// TIA Portal project "Ampelanlage" (V16)

(* hardware
DEVICE "S71500/ET200MP-Station_1"  S7-1500 station
   slot 0: "Profilschiene_0"  Rack  6ES7 590-1***0-0AA0
   slot 1: "PLC_1"  CPU 1516-3 PN/DP  6ES7 516-3AN02-0AB0  V2.8
      slot 3: "CPU-Display_1"  6ES7591-1BA00-0AA0
      slot 32768: "PROFINET-Schnittstelle_1"  X1
         slot 32769: "Port_1"  X1 P1
         slot 32770: "Port_2"  X1 P2
      slot 33024: "PROFINET-Schnittstelle_2"  X2
         slot 33025: "Port_1"  X2 P1
      slot 33280: "DP-Schnittstelle_1"  X3
      slot 34817: "Virtual CP interface port_1"  Virtual CP interface port  Virtual CP interface port
   slot 2: "DI 32x24VDC HF_1"  DI 32x24VDC HF  6ES7 521-1BL00-0AB0  V2.2
   slot 3: "DQ 32x24VDC/0.5A HF_1"  DQ 32x24VDC/0.5A HF  6ES7 522-1BL01-0AB0  V1.1
   slot 4: "AI 8xU/I/RTD/TC ST_1"  AI 8xU/I/RTD/TC ST  6ES7 531-7KF00-0AB0  V2.2
   slot 5: "AQ 4xU/I ST_1"  AQ 4xU/I ST  6ES7 532-5HD00-0AB0  V2.2
DEVICE "ET 200SP-Station_1"  ET 200SP-Station
   slot 0: "Baugruppenträger_0"  Rack  6ES5 710-8MAx1
   slot 0: "IO-Device_1"  IM 155-6 PN/2 HF  6ES7 155-6AU01-0CN0  V4.2
   slot 1: "DI 8x24VDC HF_1"  DI 8x24VDC HF  6ES7 131-6BF00-0CA0  V2.0
      slot 1: "DI 8x24VDC HF_1"  DI 8x24VDC HF
   slot 2: "DQ 8x24VDC/0.5A HF_1"  DQ 8x24VDC/0.5A HF  6ES7 132-6BF00-0CA0  V2.0
      slot 1: "DQ 8x24VDC/0.5A HF_1"  DQ 8x24VDC/0.5A HF
   slot 3: "AI 2xU/I 2-,4-wire HF_1"  AI 2xU/I 2-,4-wire HF  6ES7 134-6HB00-0CA1  V2.0
      slot 1: "AI 2xU/I 2-,4-wire HF_1"  AI 2xU/I 2-,4-wire HF
   slot 4: "AQ 2xU/I HF_1"  AQ 2xU/I HF  6ES7 135-6HB00-0CA1  V1.0
      slot 1: "AQ 2xU/I HF_1"  AQ 2xU/I HF
   slot 5: "Servermodul_1"  Server module  6ES7 193-6PA00-0AA0  V1.1
      slot 1: "Servermodul_1"  Server module
   slot 127: "BA 2xRJ45"  BA 2xRJ45  6ES7 193-6AR00-0AA0  V0.0
      slot 1: "Port_1"  X1 P1 R  6ES7 193-6AR00-0AA0  V0.0
      slot 2: "Port_2"  X1 P2 R  6ES7 193-6AR00-0AA0  V0.0
*)

// ===== PLC "PLC_1"  CPU 1516-3 PN/DP =====

VAR_GLOBAL   // PLC tag table "Ampelanlage"
   "xS0" AT %I0.0 : Bool;   // Anlage aus
   "xS7" AT %I0.7 : Bool;   // Anlage ein
   "xH0" AT %Q0.0 : Bool;   // Rot Hauptstraße
   "xH1" AT %Q0.1 : Bool;   // Gelb Hauptstraße
   "xH2" AT %Q0.2 : Bool;   // Grün Hauptsraße
   "xH3" AT %Q0.3 : Bool;   // Rot Nebenstraße
   "xH4" AT %Q0.4 : Bool;   // Gelb Nebenstraße
   "xH5" AT %Q0.5 : Bool;   // Grün Nebenstraße
   "xH6" AT %Q0.6 : Bool;   // Rot Fußgängerüberrweg
   "xH7" AT %Q0.7 : Bool;   // Grün Fußgängerüberweg
   "xS1" AT %I0.1 : Bool;   // S1 Haupt
   "xS2" AT %I0.2 : Bool;   // S2 Haupt
   "xS3" AT %I0.3 : Bool;   // S3 Neben
   "xS5" AT %I0.5 : Bool;   // S5 Fuß
   "xS6" AT %I0.6 : Bool;   // S6 Fuß
END_VAR

DATA_BLOCK "fb_Ampelanlage_DB"   // DB1
{ S7_Optimized_Access := 'TRUE' }
VERSION : 0.1
// stored: InstanceOfName fb_Ampelanlage
"fb_Ampelanlage"
BEGIN
END_DATA_BLOCK

DATA_BLOCK "fb_Ampelanlage_Bodenkontakt_DB"   // DB2
{ S7_Optimized_Access := 'TRUE' }
VERSION : 0.1
// stored: InstanceOfName fb_Ampelanlage_Bodenkontakt
"fb_Ampelanlage_Bodenkontakt"
BEGIN
END_DATA_BLOCK

FUNCTION_BLOCK "fb_Ampelanlage"   // FB1, GRAPH_PLUS
{ S7_Optimized_Access := 'TRUE' }
VERSION : 0.1
   VAR_INPUT
      OFF_SQ : Bool := false;   // Kette ausschalten
      INIT_SQ : Bool := false;   // Kette in Initialzustand versetzen
      ACK_EF : Bool := false;   // Alle Fehler und Störungen quittieren
      S_PREV : Bool := false;   // Vorherigen Schritt am Parameter S_NO ausgeben
      S_NEXT : Bool := false;   // Nächsten Schritt am Parameter S_NO anzeigen
      SW_AUTO : Bool := false;   // Automatischer Betrieb
      SW_TAP : Bool := false;   // Halbautomatisch/Weiterschalten mit Transition
      SW_TOP : Bool := false;   // Halbautomatisch/Ignoriere Transition
      SW_MAN : Bool := false;   // Handbetrieb
      S_SEL : Int := 0;   // Schritt auswählen, der an S_NO ausgegeben werden soll
      S_ON : Bool := false;   // Schritt aktivieren, der an Parameter S_NO anliegt
      S_OFF : Bool := false;   // Schritt deaktivieren, der an Parameter S_NO anliegt
      T_PUSH : Bool := false;   // Schaltfreigabe für Transition im halbautomatischen Betrieb
   END_VAR
   VAR_OUTPUT
      S_NO : Int := 0;   // Schrittnummer
      S_MORE : Bool := false;   // Weitere Schritte sind vorhanden und können in S_NO angezeigt werden.
      S_ACTIVE : Bool := false;   // Schritt, der an Parameter S_NO angezeigt wird, ist aktiv
      ERR_FLT : Bool := false;   // Sammelfehler Interlock oder Supervision
      AUTO_ON : Bool := false;   // Automatischer Betrieb eingeschaltet
      TAP_ON : Bool := false;   // Halbautomatischer Betrieb/Schritt mit Transition eingeschaltet
      TOP_ON : Bool := false;   // Halbautomatischer Betrieb/Ignoriere Transition eingeschaltet
      MAN_ON : Bool := false;   // Handbetrieb eingeschaltet
   END_VAR
   VAR
      "xTimer T1" : Bool;   // Zeit abgelaufen
      "xTimer T2" : Bool;
      "xTimer T3" : Bool;
      "xTimer T4" : Bool;
      "xTimer T5" : Bool;
      "xTimer T6" : Bool;
      "xTimer T7" : Bool;
      "xTimer T8" : Bool;
      "xTimer T9" : Bool;
      "xTimer T10" : Bool;
      HMI_INFO : Array[0..8] of UInt;
      IF_PAR : G7_IfParPlus_V6;
      RT_DATA : G7_RTDataPlus_V6;   // Interner Datenbereich
      Trans1 : G7_TransitionPlus_V6;   // Transitionsstruktur
      Trans2 : G7_TransitionPlus_V6;   // Transitionsstruktur
      Trans3 : G7_TransitionPlus_V6;   // Transitionsstruktur
      Trans4 : G7_TransitionPlus_V6;   // Transitionsstruktur
      Trans5 : G7_TransitionPlus_V6;   // Transitionsstruktur
      Trans6 : G7_TransitionPlus_V6;   // Transitionsstruktur
      Trans7 : G7_TransitionPlus_V6;   // Transitionsstruktur
      Trans8 : G7_TransitionPlus_V6;   // Transitionsstruktur
      Trans9 : G7_TransitionPlus_V6;   // Transitionsstruktur
      Step1 : G7_StepPlus_V6;   // Schrittstruktur
      Step2 : G7_StepPlus_V6;   // Schrittstruktur
      Step3 : G7_StepPlus_V6;   // Schrittstruktur
      Step4 : G7_StepPlus_V6;   // Schrittstruktur
      Step5 : G7_StepPlus_V6;   // Schrittstruktur
      Step6 : G7_StepPlus_V6;   // Schrittstruktur
      Step7 : G7_StepPlus_V6;   // Schrittstruktur
      Step8 : G7_StepPlus_V6;   // Schrittstruktur
      Step9 : G7_StepPlus_V6;   // Schrittstruktur
      SINI : Array[0..1] of USInt;
      LSTT : Array[0..8] of USInt;
      ATAJ : Array[0..8] of USInt;
      ATAB : Array[0..8] of USInt;
      PSTT : Array[0..8] of USInt;
      NSTT : Array[0..8] of USInt;
      ASSJ : Array[0..8] of USInt;
      ASSB : Array[0..8] of USInt;
      PTTS : Array[0..8] of USInt;
      NTTS : Array[0..8] of USInt;
      SW_SQTS : Array[0..8] of USInt;
      SWITCH : Array[0..0] of USInt;
      TVX : Array[0..1] of USInt;
      TTX : Array[0..1] of USInt;
      TSX : Array[0..1] of USInt;
      S00X : Array[0..1] of USInt;
      SOFFX : Array[0..1] of USInt;
      SONX : Array[0..1] of USInt;
      SAX : Array[0..1] of USInt;
      SERRX : Array[0..9] of USInt;
      SMX : Array[0..9] of USInt;
      S0X : Array[0..9] of USInt;
      S1X : Array[0..9] of USInt;
      IL_ALARM_INST : Diag_Alarm;
      SUP_ALARM_INST : Diag_Alarm;
      STEP_TIME_ALARM_INST : Diag_Alarm;
      IEC_TIMER_INST : IEC_TIMER;
      TRANSACTION_FLAG : Bool := false;
   END_VAR
   // SINI[0] := 2;
   // LSTT[0] := 255;
   // LSTT[1] := 255;
   // LSTT[2] := 255;
   // LSTT[3] := 255;
   // LSTT[4] := 255;
   // LSTT[5] := 255;
   // LSTT[6] := 255;
   // LSTT[7] := 255;
   // ATAJ[1] := 1;
   // ATAJ[2] := 2;
   // ATAJ[3] := 3;
   // ATAJ[4] := 4;
   // ATAJ[5] := 5;
   // ATAJ[6] := 6;
   // ATAJ[7] := 7;
   // ATAJ[8] := 8;
   // ATAB[1] := 1;
   // ATAB[2] := 2;
   // ATAB[3] := 3;
   // ATAB[4] := 4;
   // ATAB[5] := 5;
   // ATAB[6] := 6;
   // ATAB[7] := 7;
   // ATAB[8] := 8;
   // PSTT[1] := 1;
   // PSTT[2] := 2;
   // PSTT[3] := 3;
   // PSTT[4] := 4;
   // PSTT[5] := 5;
   // PSTT[6] := 6;
   // PSTT[7] := 7;
   // PSTT[8] := 8;
   // NSTT[0] := 1;
   // NSTT[1] := 2;
   // NSTT[2] := 3;
   // NSTT[3] := 4;
   // NSTT[4] := 5;
   // NSTT[5] := 6;
   // NSTT[6] := 7;
   // NSTT[7] := 8;
   // ASSJ[1] := 1;
   // ASSJ[2] := 2;
   // ASSJ[3] := 3;
   // ASSJ[4] := 4;
   // ASSJ[5] := 5;
   // ASSJ[6] := 6;
   // ASSJ[7] := 7;
   // ASSJ[8] := 8;
   // ASSB[1] := 1;
   // ASSB[2] := 2;
   // ASSB[3] := 3;
   // ASSB[4] := 4;
   // ASSB[5] := 5;
   // ASSB[6] := 6;
   // ASSB[7] := 7;
   // ASSB[8] := 8;
   // PTTS[0] := 255;
   // PTTS[2] := 1;
   // PTTS[3] := 2;
   // PTTS[4] := 3;
   // PTTS[5] := 4;
   // PTTS[6] := 5;
   // PTTS[7] := 6;
   // PTTS[8] := 7;
   // NTTS[1] := 1;
   // NTTS[2] := 2;
   // NTTS[3] := 3;
   // NTTS[4] := 4;
   // NTTS[5] := 5;
   // NTTS[6] := 6;
   // NTTS[7] := 7;
   // NTTS[8] := 8;
   // TVX[0] := 16#1;
   // TTX[0] := 16#1;
   // TSX[0] := 16#1;
   // S00X[0] := 16#1;
   // SOFFX[0] := 16#1;
   // SONX[0] := 16#1;
   // SAX[0] := 16#1;
   // SERRX[0] := 16#1;
   // SMX[0] := 16#1;
   // S0X[0] := 16#1;
   // S1X[0] := 16#1;
BEGIN
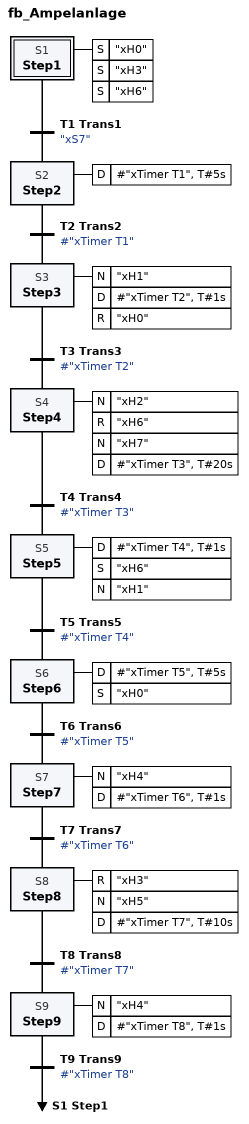
   // sequencer 1
   INITIAL_STEP Step1:   // S1, max time T#10S, warning time T#7S
      // Alle Ampeln Rot
              S    "xH0"
              S    "xH3"
              S    "xH6"
   END_STEP
   TRANSITION Trans1 FROM Step1 TO Step2   // T1
      := "xS7";
   END_TRANSITION
   STEP Step2:   // S2, max time T#10S, warning time T#7S
              D    #"xTimer T1", T#5s
   END_STEP
   TRANSITION Trans2 FROM Step2 TO Step3   // T2
      := #"xTimer T1";
   END_TRANSITION
   STEP Step3:   // S3, max time T#10S, warning time T#7S
              N    "xH1"
              D    #"xTimer T2", T#1s
              R    "xH0"
   END_STEP
   TRANSITION Trans3 FROM Step3 TO Step4   // T3
      := #"xTimer T2";
   END_TRANSITION
   STEP Step4:   // S4, max time T#10S, warning time T#7S
              N    "xH2"
              R    "xH6"
              N    "xH7"
              D    #"xTimer T3", T#20s
   END_STEP
   TRANSITION Trans4 FROM Step4 TO Step5   // T4
      := #"xTimer T3";
   END_TRANSITION
   STEP Step5:   // S5, max time T#10S, warning time T#7S
              D    #"xTimer T4", T#1s
              S    "xH6"
              N    "xH1"
   END_STEP
   TRANSITION Trans5 FROM Step5 TO Step6   // T5
      := #"xTimer T4";
   END_TRANSITION
   STEP Step6:   // S6, max time T#10S, warning time T#7S
              D    #"xTimer T5", T#5s
              S    "xH0"
   END_STEP
   TRANSITION Trans6 FROM Step6 TO Step7   // T6
      := #"xTimer T5";
   END_TRANSITION
   STEP Step7:   // S7, max time T#10S, warning time T#7S
              N    "xH4"
              D    #"xTimer T6", T#1s
   END_STEP
   TRANSITION Trans7 FROM Step7 TO Step8   // T7
      := #"xTimer T6";
   END_TRANSITION
   STEP Step8:   // S8, max time T#10S, warning time T#7S
              R    "xH3"
              N    "xH5"
              D    #"xTimer T7", T#10s
   END_STEP
   TRANSITION Trans8 FROM Step8 TO Step9   // T8
      := #"xTimer T7";
   END_TRANSITION
   STEP Step9:   // S9, max time T#10S, warning time T#7S
              N    "xH4"
              D    #"xTimer T8", T#1s
   END_STEP
   TRANSITION Trans9 FROM Step9 TO Step1   // T9, jump
      := #"xTimer T8";
   END_TRANSITION
END_FUNCTION_BLOCK

FUNCTION_BLOCK "fb_Ampelanlage_Bodenkontakt"   // FB2, GRAPH_PLUS
{ S7_Optimized_Access := 'TRUE' }
VERSION : 0.1
   VAR_INPUT
      OFF_SQ : Bool := false;   // Kette ausschalten
      INIT_SQ : Bool := false;   // Kette in Initialzustand versetzen
      ACK_EF : Bool := false;   // Alle Fehler und Störungen quittieren
      S_PREV : Bool := false;   // Vorherigen Schritt am Parameter S_NO ausgeben
      S_NEXT : Bool := false;   // Nächsten Schritt am Parameter S_NO anzeigen
      SW_AUTO : Bool := false;   // Automatischer Betrieb
      SW_TAP : Bool := false;   // Halbautomatisch/Weiterschalten mit Transition
      SW_TOP : Bool := false;   // Halbautomatisch/Ignoriere Transition
      SW_MAN : Bool := false;   // Handbetrieb
      S_SEL : Int := 0;   // Schritt auswählen, der an S_NO ausgegeben werden soll
      S_ON : Bool := false;   // Schritt aktivieren, der an Parameter S_NO anliegt
      S_OFF : Bool := false;   // Schritt deaktivieren, der an Parameter S_NO anliegt
      T_PUSH : Bool := false;   // Schaltfreigabe für Transition im halbautomatischen Betrieb
   END_VAR
   VAR_OUTPUT
      S_NO : Int := 0;   // Schrittnummer
      S_MORE : Bool := false;   // Weitere Schritte sind vorhanden und können in S_NO angezeigt werden.
      S_ACTIVE : Bool := false;   // Schritt, der an Parameter S_NO angezeigt wird, ist aktiv
      ERR_FLT : Bool := false;   // Sammelfehler Interlock oder Supervision
      AUTO_ON : Bool := false;   // Automatischer Betrieb eingeschaltet
      TAP_ON : Bool := false;   // Halbautomatischer Betrieb/Schritt mit Transition eingeschaltet
      TOP_ON : Bool := false;   // Halbautomatischer Betrieb/Ignoriere Transition eingeschaltet
      MAN_ON : Bool := false;   // Handbetrieb eingeschaltet
   END_VAR
   VAR
      "xTimer T2" : Bool;
      "xTimer T1" : Bool;
      "xTimer T4" : Bool;
      "xTimer T5" : Bool;
      "xTimer T7" : Bool;
      "xTimer T6" : Bool;
      "xTimer T8" : Bool;
      "xTimer T9" : Bool;
      "xTimer T10" : Bool;
      "xTimer T3" : Bool;
      HMI_INFO : Array[0..8] of UInt;
      IF_PAR : G7_IfParPlus_V6;
      RT_DATA : G7_RTDataPlus_V6;   // Interner Datenbereich
      Trans1 : G7_TransitionPlus_V6;   // Transitionsstruktur
      Trans2 : G7_TransitionPlus_V6;   // Transitionsstruktur
      Trans3 : G7_TransitionPlus_V6;   // Transitionsstruktur
      Trans4 : G7_TransitionPlus_V6;   // Transitionsstruktur
      Trans5 : G7_TransitionPlus_V6;   // Transitionsstruktur
      Trans13 : G7_TransitionPlus_V6;   // Transitionsstruktur
      Trans101 : G7_TransitionPlus_V6;   // Transitionsstruktur
      Trans7 : G7_TransitionPlus_V6;   // Transitionsstruktur
      Trans8 : G7_TransitionPlus_V6;   // Transitionsstruktur
      Trans9 : G7_TransitionPlus_V6;   // Transitionsstruktur
      Trans10 : G7_TransitionPlus_V6;   // Transitionsstruktur
      Trans11 : G7_TransitionPlus_V6;   // Transitionsstruktur
      Step1 : G7_StepPlus_V6;   // Schrittstruktur
      Step2 : G7_StepPlus_V6;   // Schrittstruktur
      Step3 : G7_StepPlus_V6;   // Schrittstruktur
      Step4 : G7_StepPlus_V6;   // Schrittstruktur
      Step5 : G7_StepPlus_V6;   // Schrittstruktur
      Step204 : G7_StepPlus_V6;   // Schrittstruktur
      Step7 : G7_StepPlus_V6;   // Schrittstruktur
      Step8 : G7_StepPlus_V6;   // Schrittstruktur
      Step9 : G7_StepPlus_V6;   // Schrittstruktur
      Step10 : G7_StepPlus_V6;   // Schrittstruktur
      SINI : Array[0..1] of USInt;
      LSTT : Array[0..11] of USInt;
      ATAJ : Array[0..11] of USInt;
      ATAB : Array[0..11] of USInt;
      PSTT : Array[0..11] of USInt;
      NSTT : Array[0..11] of USInt;
      ASSJ : Array[0..9] of USInt;
      ASSB : Array[0..9] of USInt;
      PTTS : Array[0..9] of USInt;
      NTTS : Array[0..9] of USInt;
      SW_SQTS : Array[0..9] of USInt;
      SWITCH : Array[0..1] of USInt;
      TVX : Array[0..4] of USInt;
      TTX : Array[0..4] of USInt;
      TSX : Array[0..1] of USInt;
      S00X : Array[0..1] of USInt;
      SOFFX : Array[0..1] of USInt;
      SONX : Array[0..1] of USInt;
      SAX : Array[0..1] of USInt;
      SERRX : Array[0..10] of USInt;
      SMX : Array[0..10] of USInt;
      S0X : Array[0..10] of USInt;
      S1X : Array[0..10] of USInt;
      IL_ALARM_INST : Diag_Alarm;
      SUP_ALARM_INST : Diag_Alarm;
      STEP_TIME_ALARM_INST : Diag_Alarm;
      IEC_TIMER_INST : IEC_TIMER;
      TRANSACTION_FLAG : Bool := false;
   END_VAR
   // SINI[0] := 2;
   // LSTT[0] := 255;
   // LSTT[1] := 255;
   // LSTT[2] := 255;
   // LSTT[3] := 255;
   // LSTT[5] := 255;
   // LSTT[7] := 255;
   // LSTT[8] := 255;
   // LSTT[9] := 255;
   // LSTT[10] := 255;
   // ATAJ[1] := 1;
   // ATAJ[2] := 2;
   // ATAJ[3] := 3;
   // ATAJ[4] := 4;
   // ATAJ[5] := 5;
   // ATAJ[6] := 6;
   // ATAJ[7] := 7;
   // ATAJ[8] := 8;
   // ATAJ[9] := 9;
   // ATAJ[10] := 10;
   // ATAJ[11] := 11;
   // ATAB[0] := 5;
   // ATAB[1] := 1;
   // ATAB[2] := 2;
   // ATAB[3] := 3;
   // ATAB[4] := 4;
   // ATAB[5] := 7;
   // ATAB[6] := 6;
   // ATAB[8] := 8;
   // ATAB[9] := 9;
   // ATAB[10] := 10;
   // ATAB[11] := 11;
   // PSTT[1] := 1;
   // PSTT[2] := 2;
   // PSTT[3] := 3;
   // PSTT[4] := 4;
   // PSTT[6] := 5;
   // PSTT[8] := 6;
   // PSTT[9] := 7;
   // PSTT[10] := 8;
   // PSTT[11] := 9;
   // NSTT[0] := 1;
   // NSTT[1] := 2;
   // NSTT[2] := 3;
   // NSTT[3] := 4;
   // NSTT[5] := 5;
   // NSTT[7] := 6;
   // NSTT[8] := 7;
   // NSTT[9] := 8;
   // NSTT[10] := 9;
   // ASSJ[1] := 1;
   // ASSJ[2] := 2;
   // ASSJ[3] := 3;
   // ASSJ[4] := 4;
   // ASSJ[5] := 5;
   // ASSJ[6] := 6;
   // ASSJ[7] := 7;
   // ASSJ[8] := 8;
   // ASSJ[9] := 9;
   // ASSB[1] := 1;
   // ASSB[2] := 2;
   // ASSB[3] := 3;
   // ASSB[4] := 4;
   // ASSB[5] := 5;
   // ASSB[6] := 6;
   // ASSB[7] := 7;
   // ASSB[8] := 8;
   // ASSB[9] := 9;
   // PTTS[0] := 255;
   // PTTS[2] := 1;
   // PTTS[3] := 2;
   // PTTS[4] := 3;
   // PTTS[5] := 5;
   // PTTS[6] := 7;
   // PTTS[7] := 8;
   // PTTS[8] := 9;
   // PTTS[9] := 10;
   // NTTS[1] := 1;
   // NTTS[2] := 2;
   // NTTS[3] := 3;
   // NTTS[4] := 4;
   // NTTS[5] := 6;
   // NTTS[6] := 8;
   // NTTS[7] := 9;
   // NTTS[8] := 10;
   // NTTS[9] := 11;
   // SW_SQTS[1] := 1;
   // SW_SQTS[2] := 1;
   // SW_SQTS[3] := 1;
   // SW_SQTS[4] := 1;
   // SW_SQTS[5] := 2;
   // SW_SQTS[6] := 3;
   // SW_SQTS[7] := 3;
   // SW_SQTS[8] := 3;
   // SW_SQTS[9] := 3;
   // TVX[0] := 16#1;
   // TTX[0] := 16#1;
   // TSX[0] := 16#1;
   // S00X[0] := 16#1;
   // SOFFX[0] := 16#1;
   // SONX[0] := 16#1;
   // SAX[0] := 16#1;
   // SERRX[0] := 16#1;
   // SMX[0] := 16#1;
   // S0X[0] := 16#1;
   // S1X[0] := 16#1;
BEGIN
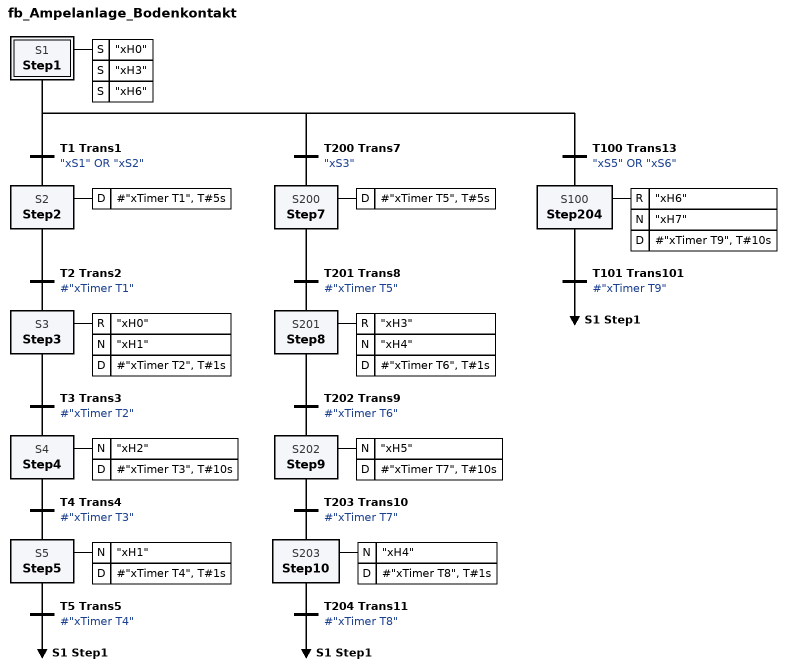
   // sequencer 1
   INITIAL_STEP Step1:   // S1, max time T#10S, warning time T#7S
      // Alle Ampeln rot
              S    "xH0"
              S    "xH3"
              S    "xH6"
   END_STEP
   TRANSITION Trans1 FROM Step1 TO Step2   // T1
      := "xS1" OR "xS2";
   END_TRANSITION
   TRANSITION Trans7 FROM Step1 TO Step7   // T200
      := "xS3";
   END_TRANSITION
   TRANSITION Trans13 FROM Step1 TO Step204   // T100
      := "xS5" OR "xS6";
   END_TRANSITION
   STEP Step2:   // S2, max time T#10S, warning time T#7S
              D    #"xTimer T1", T#5s
   END_STEP
   TRANSITION Trans2 FROM Step2 TO Step3   // T2
      := #"xTimer T1";
   END_TRANSITION
   STEP Step3:   // S3, max time T#10S, warning time T#7S
              R    "xH0"
              N    "xH1"
              D    #"xTimer T2", T#1s
   END_STEP
   TRANSITION Trans3 FROM Step3 TO Step4   // T3
      := #"xTimer T2";
   END_TRANSITION
   STEP Step4:   // S4, max time T#10S, warning time T#7S
              N    "xH2"
              D    #"xTimer T3", T#10s
   END_STEP
   TRANSITION Trans4 FROM Step4 TO Step5   // T4
      := #"xTimer T3";
   END_TRANSITION
   STEP Step5:   // S5, max time T#10S, warning time T#7S
              N    "xH1"
              D    #"xTimer T4", T#1s
   END_STEP
   TRANSITION Trans5 FROM Step5 TO Step1   // T5, jump
      := #"xTimer T4";
   END_TRANSITION
   STEP Step8:   // S201, max time T#10S, warning time T#7S
              R    "xH3"
              N    "xH4"
              D    #"xTimer T6", T#1s
   END_STEP
   TRANSITION Trans9 FROM Step8 TO Step9   // T202
      := #"xTimer T6";
   END_TRANSITION
   STEP Step7:   // S200, max time T#10S, warning time T#7S
              D    #"xTimer T5", T#5s
   END_STEP
   TRANSITION Trans8 FROM Step7 TO Step8   // T201
      := #"xTimer T5";
   END_TRANSITION
   STEP Step9:   // S202, max time T#10S, warning time T#7S
              N    "xH5"
              D    #"xTimer T7", T#10s
   END_STEP
   TRANSITION Trans10 FROM Step9 TO Step10   // T203
      := #"xTimer T7";
   END_TRANSITION
   STEP Step10:   // S203, max time T#10S, warning time T#7S
              N    "xH4"
              D    #"xTimer T8", T#1s
   END_STEP
   TRANSITION Trans11 FROM Step10 TO Step1   // T204, jump
      := #"xTimer T8";
   END_TRANSITION
   STEP Step204:   // S100, max time T#10S, warning time T#7S
              R    "xH6"
              N    "xH7"
              D    #"xTimer T9", T#10s
   END_STEP
   TRANSITION Trans101 FROM Step204 TO Step1   // T101, jump
      := #"xTimer T9";
   END_TRANSITION
END_FUNCTION_BLOCK

ORGANIZATION_BLOCK "Main"   // OB1, FBD, ProgramCycle
TITLE = "Main Program Sweep (Cycle)"
{ S7_Optimized_Access := 'TRUE' }
VERSION : 0.1
   VAR_INPUT
      Initial_Call : Bool;   // Initial call of this OB
      Remanence : Bool;   // =True, if remanent data are available
   END_VAR
BEGIN

REGION Network 1
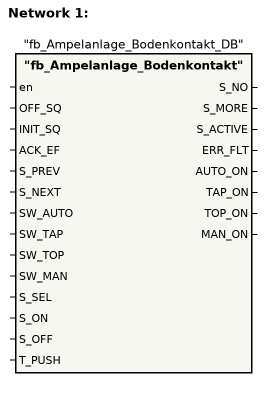
   "fb_Ampelanlage_Bodenkontakt_DB"();   // "fb_Ampelanlage_Bodenkontakt"
END_REGION
END_ORGANIZATION_BLOCK